# EPICS substitutions: db/ecmcEK1100.substitutions
file ecmcEcSlave.template
{
    pattern {}
            {}
}
